TYPE ZDataConfig :
STRUCT
{region "Handling"}
{IF NOT (defined (Handling_disabled))}
  Handling : HandlingDataConfig;
  {attribute 'ZId' := 'a0dd13f9-743a-4c3b-9b43-ecc916834d10'}
{END_IF}
{endregion}
{region "Mover1"}
{IF NOT (defined (Mover1_disabled))}
  Mover1 : MoverDataConfig;
  {attribute 'ZId' := '0635b537-20e6-40de-ab4b-39921311b510'}
{END_IF}
{endregion}
{attribute '__ZwPlcApplicationDataConfigDeclaration__'} // Do not remove this attribute! It is used for code generation.
END_STRUCT
END_TYPE

(* stored: Version 1.1.0.1
   DUT ZDataConfig: Id {7cd3b5b4-ed66-4b4f-8ead-56478cfcf810} *)
